{attribute addProperty BoxType "AT2000-0233-0022"}
{attribute addProperty Id "CC_Inputs_14_ChAT %I*CC_Inputs_14_Ch_5FB71CBE240300CC_Outputs_14_ChAT %Q*CC_Outputs_14_Ch_8D55E481240300WcStateAT %I*WcState_F855686C1620InfoDataAT %I*InfoData_0BDED7BF144180"}
{attribute addProperty CRC "517270396"}
{attribute addProperty SizeInBites "640"}
{attribute addProperty SizeInBytes "80"}
TYPE AT2000_050BA888 :
STRUCT
	{attribute addProperty Name "CC_Inputs_14_Ch"}
	CC_Inputs_14_Ch : CC_Inputs_14_Ch_5FB71CBE;
	{attribute addProperty Name "CC_Outputs_14_Ch"}
	CC_Outputs_14_Ch : CC_Outputs_14_Ch_8D55E481;
	{attribute addProperty Name "WcState"}
	WcState : WcState_F855686C;
	{attribute addProperty Name "InfoData"}
	InfoData : InfoData_0BDED7BF;
END_STRUCT
END_TYPE

(* stored: Version 1.2.0.0, ProductVersion 3.1.4024.9
   DUT AT2000_050BA888: Id {edb78f3c-9bc1-4f64-bfc6-7627f7c8600b} *)
